SUBAPPLICATION Uebung_012f (* Numeric Value Input PHYS und Speichern NVS mit Subapp *)
  (* Standard: 61499-2; Description: Copyright (c) 2023 Meisterschulen am Ostbahnhof This program and the accompanying materials are made available under the terms of the Eclipse Public License 2.0 which is available at https://www.eclipse.org/legal/epl-2.0/ SPDX-License-Identifier: EPL-2.0 *)
  (* Version 1.0, 2023-10-23, Franz Höpfinger, Meisterschulen am Ostbahnhof, initial API and implementation and/or initial documentation *)
  PACKAGE Uebungen;
  IMPORT Uebungen::const::NVS::NVS_Keys::KEY_I1_STORE;
  IMPORT Uebungen::const::UT::DefaultPool_Numeric::InputNumber_I1_N;
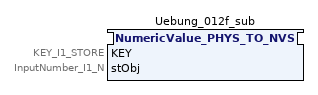
  SUBAPPS
    Uebung_012f_sub : MyLib::sys::NumericValue_PHYS_TO_NVS(KEY := KEY_I1_STORE, stObj := InputNumber_I1_N);
  END_SUBAPPS
END_SUBAPPLICATION
